Staubli VAL3: JudgeSpace.pgx

public program JudgeSpace(num& x_nRes, string x_sStrIn)
  local num l_i
begin
  //判断一个字符串是否是空格字符串
  //x_nRes=0:非空格字符串
  //x_nRes=1:空格字符串
  //x_nRes=2:空字符串
  x_nRes=0
  if x_sStrIn==""
    x_nRes=2
    return
  endIf
  for l_i=0 to len(x_sStrIn)-1
    if left(x_sStrIn,1)==" "
      x_sStrIn=right(x_sStrIn,len(x_sStrIn)-1)
    else
      return
    endIf
  endFor
  x_nRes=1
end
